FUNCTION_BLOCK FB_CSVPersistentEventStorage IMPLEMENTS I_PersistentStorage

VAR
	
	fileOpen: FB_FileOpen:=(sPathName:='c:\Events.log',nMode:= FOPEN_MODEAPPEND OR FOPEN_MODETEXT );
	fileClose: FB_FileClose;
	filePuts: FB_FilePuts;
	eWriteState: (FILE_OPEN_TRIGGER,FILE_OPEN, WAIT_FOR_EVENT, WRITE_EVENT_TRIGGER,WRITE_EVENT, FILE_CLOSE_TRIGGER, FILE_CLOSE, ERROR);
	stEventWrittenToFile: ST_Event;
	
	CsvString:T_MaxString;
	
END_VAR

CASE eWriteState OF
	FILE_OPEN_TRIGGER:
				fileOpen(bExecute:=TRUE);
				eWriteState:= FILE_OPEN;
	FILE_OPEN:
				fileOpen(bExecute:=FALSE);
				IF fileOpen.bError THEN
					eWriteState:= ERROR;
				ELSIF NOT fileOpen.bBusy AND fileOpen.hFile <> 0 THEN
					eWriteState := WAIT_FOR_EVENT;		
				END_IF
	WAIT_FOR_EVENT:
		//Do Nothing
	WRITE_EVENT_TRIGGER:
		CsvString := CreateCsvString(stEvent:=stEventWrittenToFile);
		
		filePuts(bExecute:= TRUE, sLine:=CsvString,hFile:=fileOpen.hFile );
		eWriteState := WRITE_EVENT;
				
	WRITE_EVENT:
			filePuts(bExecute:=FALSE);
			IF filePuts.bError THEN
					eWriteState:= ERROR;
				ELSIF NOT filePuts.bBusy  THEN
					eWriteState := FILE_CLOSE_TRIGGER;		
				END_IF
	FILE_CLOSE_TRIGGER:
		fileClose(bExecute:=TRUE,hFile:=fileOpen.hFile);
				eWriteState := FILE_CLOSE;
	FILE_CLOSE:
		fileClose(bExecute:=FALSE);
		IF fileClose.bError THEN
			eWriteState:= ERROR;
		ELSIF NOT fileClose.bBusy THEN
			eWriteState:=	FILE_OPEN_TRIGGER;
		END_IF
	ERROR:
	//Error Code here
	
END_CASE

METHOD CreateCsvString : T_MaxString
VAR_INPUT
	stEvent: REFERENCE TO ST_Event;
	
END_VAR
VAR
	Tempstring: T_MaxString;
END_VAR
Tempstring:= TO_STRING(stEvent.eEventType);
Tempstring:=CONCAT(STR1:= Tempstring, STR2:= ',');
Tempstring:=CONCAT(STR1:= Tempstring, STR2:= TO_STRING(stEvent.eEventSeverity));
Tempstring:=CONCAT(STR1:= Tempstring, STR2:= ',');
Tempstring:=CONCAT(STR1:= Tempstring, STR2:= TO_STRING(stEvent.nEventIdentity));
Tempstring:=CONCAT(STR1:= Tempstring, STR2:= ',');
Tempstring:=CONCAT(STR1:= Tempstring, STR2:= TO_STRING(stEvent.sEventText));
Tempstring:=CONCAT(STR1:= Tempstring, STR2:= ',');
Tempstring:=CONCAT(STR1:= Tempstring, STR2:= TO_STRING(stEvent.dtTimeStamp));
Tempstring:=CONCAT(STR1:= Tempstring, STR2:= '$n');

CreateCsvString:= Tempstring;
END_METHOD

{warning 'add method implementation '}
METHOD StoreEvent
VAR_INPUT
	stEvent	: ST_Event;
END_VAR
//Implement code here
IF eWriteState =  WAIT_FOR_EVENT THEN
	eWriteState:= WRITE_EVENT_TRIGGER;
	stEventWrittenToFile:=stEvent;

END_IF
END_METHOD

END_FUNCTION_BLOCK

(* stored: Version 1.1.0.1, ProductVersion 3.1.4024.11
   POU FB_CSVPersistentEventStorage: Id {48057f67-f8f3-456e-8b98-5d8825e7cf1e}, SpecialFunc None
   Method CreateCsvString: Id {1667a629-d2bb-454b-9b8e-5ea3a3f673ac}
   Method StoreEvent: Id {96bacc2c-21ac-45b8-8511-0845dc5a77db} *)
